// TIA Portal V20 export
TYPE "LER_typeAlignSyncMoveCommands"
// stored: Access Published
   STRUCT
      MoveCw : Bool;
      MoveCcw : Bool;
      MoveYPlus : Bool;
      MoveYMinus : Bool;
      errorAck : Bool;
   END_STRUCT;
END_TYPE
